TYPE TYP_VESSEL_HW_IN :
STRUCT
	Sensor : REAL; //pressure of the vessel
END_STRUCT
END_TYPE

(* stored: Version 1.1.0.1, ProductVersion 3.1.4024.12
   DUT TYP_VESSEL_HW_IN: Id {9dfff377-773b-4386-aac4-95bf5ef3c506} *)
